FUNCTION_BLOCK Hutschienenmoped_3_DI_DOUBLE_CLICK (* Service Interface Function Block Type *)
  (* Function: All Inputs; Description: this maps to IE *)
  (* Version 1.0, 2018-12-05, Jose Cabral *)
  (* Version 1.1, 2022-08-04, Franz Höpfinger, HR Agrartechnik GmbH *)
  (* Version 1.2, 2023-01-05, Franz Höpfinger, HR Agrartechnik GmbH *)
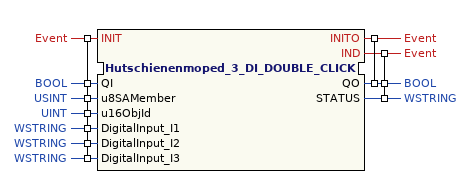
  EVENT_INPUT
    INIT WITH QI, u8SAMember, u16ObjId, DigitalInput_I1, DigitalInput_I2, DigitalInput_I3; (* Service Initialization *)
  END_EVENT
  EVENT_OUTPUT
    INITO WITH QO; (* Initialization Confirm *)
    IND WITH QO, STATUS; (* Indication from Resource *)
  END_EVENT
  VAR_INPUT
    QI : BOOL; (* Event Input Qualifier *)
    u8SAMember : USINT := 255; (* Dummy !, set to 255 if in doubt. 0 deactivates FB. *)
    u16ObjId : UINT := 65535; (* Dummy ! set to 65535 if in Doubt. 0 deactivates FB. *)
    DigitalInput_I1 : WSTRING := "DigitalInput_I1_DOUBLE_CLICK"; (* Identifier for Input 1 *)
    DigitalInput_I2 : WSTRING := "DigitalInput_I2_DOUBLE_CLICK"; (* Identifier for Input 2 *)
    DigitalInput_I3 : WSTRING := "DigitalInput_I3_DOUBLE_CLICK"; (* Identifier for Input 3 *)
  END_VAR
  VAR_OUTPUT
    QO : BOOL; (* Event Output Qualifier *)
    STATUS : WSTRING; (* Service Status *)
  END_VAR
END_FUNCTION_BLOCK
